// Mitsubishi GX Works2 project: 0715점프FEND   PLC: Q02/Q02H

PROGRAM MAIN
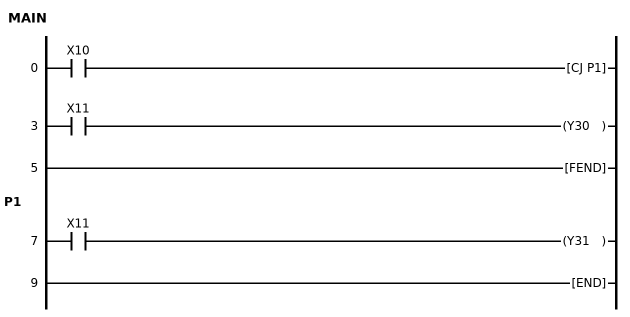
0     LD      X10
      CJ      P1
3     LD      X11
      OUT     Y30
5     FEND
      P1
7     LD      X11
      OUT     Y31
9     END
END_PROGRAM
